FUNCTION_BLOCK {name} (* {name} Function Block Type *)
  (* Standard: 61499-2 *)
  (* Version 0.1, {date}, {author}, NetAllied *)
  (* Compiler header: package fb.rt.template; *)
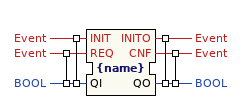
  EVENT_INPUT
    INIT WITH QI; (* Initialization Request *)
    REQ WITH QI; (* Normal Execution Request *)
  END_EVENT
  EVENT_OUTPUT
    INITO WITH QO; (* Initialization Confirm *)
    CNF WITH QO; (* Execution Confirmation *)
  END_EVENT
  VAR_INPUT
    QI : BOOL; (* Input event qualifier *)
  END_VAR
  VAR_OUTPUT
    QO : BOOL; (* Output event qualifier *)
  END_VAR
  EC_STATES
    START; (* Initial State *)
  END_STATES
  ALGORITHM INIT IN ST: (* Init algorithm *)

  END_ALGORITHM
END_FUNCTION_BLOCK
